PROGRAM CoffeeMaker

VAR
	CoffeeTimer : TON; // Timer for making coffee
END_VAR

IF (GVL.bAlarmON AND GVL.bLightsON) THEN
	CoffeeTimer(IN := TRUE, PT := GVL.tCoffeeTime); //Starting the timer for 15 seconds
ELSE
	CoffeeTimer(IN := FALSE);
	GVL.bCoffeeReady := FALSE;
END_IF

IF CoffeeTimer.Q THEN
	GVL.bCoffeeReady := TRUE;
END_IF

END_PROGRAM

(* stored: Version 1.1.0.1, ProductVersion 3.1.4024.12
   POU CoffeeMaker: Id {e1d1c9b2-a77c-40e4-84be-22e4d616f582}, SpecialFunc None *)
